PROGRAM P_Demo_F_BA_WeekNDayVal
VAR
    argEWeekday                    : E_BA_Weekday                  ; // eWeekday
    argEWeekOfMonth                : E_BA_Week                     ; // eWeekOfMonth
    argEMonth                      : E_BA_Month                    ; // eMonth
    fnReturn                       : U_BA_DateVal; // 返回值
END_VAR

// =============================================================================
// Tc3_BA2_Common.F_BA_WeekNDayVal 演示程序
// =============================================================================
// 场景："每月第二个星期日为夏令时切换" —— 把 WeekNDay 打包供调度引擎。
//
// 价值：同上：统一接口让调度引擎处理。
//
// 验证：登录 PLC 后，按例程内变量在线写值；监视输出 / 返回值，结合 §1 功能
//       简述的预期行为对照（详见配套 .md 文档 §7 业务场景）。
//
// 验证步骤：
//   1. 右键 PLC 项目下 POUs 文件夹 → Add → Existing Item → 选本 .TcPOU 文件
//   2. 引用 Tc3_BA2_Common（References → Add library）
//   3. 编译 → 登录 → 运行；按上方『验证』指引在线写值观察
// =============================================================================

fnReturn := F_BA_WeekNDayVal(
    eWeekday                 := argEWeekday,
    eWeekOfMonth             := argEWeekOfMonth,
    eMonth                   := argEMonth
);

END_PROGRAM

(* stored: Version 1.1.0.1, ProductVersion 3.1.4024.5
   POU P_Demo_F_BA_WeekNDayVal: Id {603e4b7b-2f5b-55bf-bc40-d69dbad5d28d}, SpecialFunc None *)
